(*
SPDX-FileCopyrightText: © 2026 Oleksandr Tiutyk <trofimich@gmail.com>
SPDX-License-Identifier: MIT
License: https://opensource.org/license/mit
*)

{attribute 'no_explicit_call' := 'do not call this POU directly'}
PROGRAM INTERNAL CurrentNamespace
VAR
	{attribute 'hide'} 
	_NamespaceExtractor : NamespaceExtractor;
END_VAR

{attribute 'monitoring' := 'call'}
PROPERTY Name : REFERENCE TO STRING
GET
Name REF= _NamespaceExtractor.CurrentNamespace;
END_GET
END_PROPERTY

END_PROGRAM

(* stored: Version 1.1.0.1
   POU CurrentNamespace: Id {15b1621d-0ca4-4335-9fb3-a6b21ffefa44}, SpecialFunc None
   Property Name: Id {8860504b-f01c-4478-804e-524a841d9f33}
   Get Get: Id {d82093b1-a7e1-403e-adff-5be5bedf926f} *)
